ABB RobotStudio station: Proyecto.rsstn

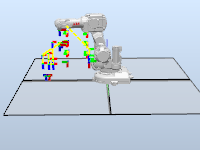
Station Proyecto (saved by RobotStudio 22.1.9826.0)
Controller IRB140_6_81
  mechanical unit ROB_1: IRB140_6_81_C_03_2, 6 joints, base frame (0, 0, 0) mm
Layout (positions relative to the parent item):
  - IRB140_6_81_C_03_2 [mechanism, from Robots\IRB140_6_81_C_G_03.rslib] at (0, 0, 0) mm; joint values [0.0983, 0.2535, -0.224, 0, 1.5413, 0.0983] (rad or m)
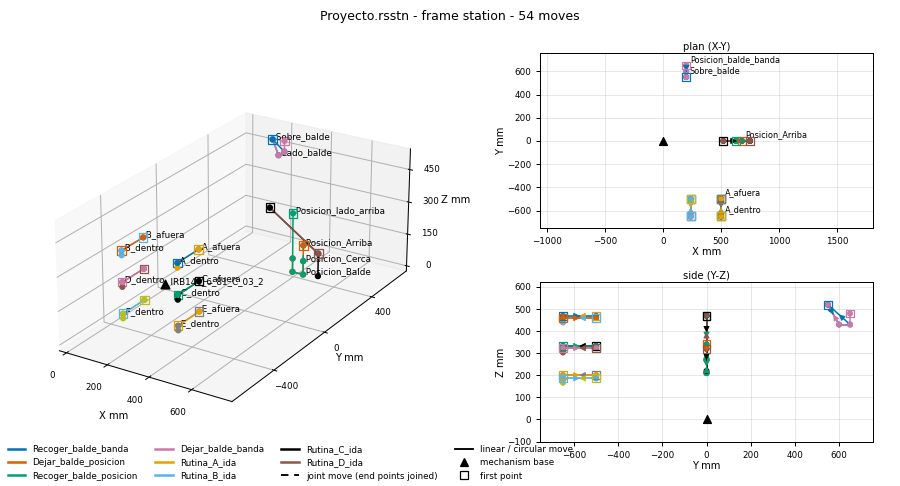
[picture p0: tool path of Proyecto.rsstn in frame station, 54 of 57 moves have a stored position in this frame; points joined in program order, loops and branches not executed]
Targets, tools, work objects and paths stored in the station, written as RAPID:
! task T_ROB1
MODULE Module1
  CONST jointtarget Home:=[[0,0,0,0,0,0],[9E+09,9E+09,9E+09,9E+09,9E+09,9E+09]];
  CONST robtarget Sobre_balde:=[[-100,0,-100],[0.707106781,0,0.707106781,0],[0,0,0,0],[9E+09,9E+09,9E+09,9E+09,9E+09,9E+09]];
  CONST robtarget Lado_balde:=[[-10,0,-50],[0.707106781,0,0.707106781,0],[0,0,-1,0],[9E+09,9E+09,9E+09,9E+09,9E+09,9E+09]];
  CONST robtarget Posicion_balde_banda:=[[-10,0,0],[0.707106781,0,0.707106781,0],[0,0,-1,0],[9E+09,9E+09,9E+09,9E+09,9E+09,9E+09]];
  CONST robtarget Dejando_balde:=[[-60,0,0],[0.707106781,0,0.707106781,0],[0,0,-1,0],[9E+09,9E+09,9E+09,9E+09,9E+09,9E+09]];
  CONST robtarget Posicion_Arriba:=[[-270,0,0],[0.707106781,0,0.707106781,0],[-1,1,-2,0],[9E+09,9E+09,9E+09,9E+09,9E+09,9E+09]];
  CONST robtarget Posicion_Cerca:=[[-200,0,0],[0.707106781,0,0.707106781,0],[-1,1,-2,0],[9E+09,9E+09,9E+09,9E+09,9E+09,9E+09]];
  CONST robtarget Posicion_Balde:=[[-140,0,0],[0.707106781,0,0.707106781,0],[-1,1,-2,0],[9E+09,9E+09,9E+09,9E+09,9E+09,9E+09]];
  CONST robtarget Posicion_lado:=[[-140,0,-50],[0.707106781,0,0.707106781,0],[-1,1,-2,0],[9E+09,9E+09,9E+09,9E+09,9E+09,9E+09]];
  CONST robtarget Posicion_lado_cerca:=[[-200,0,-50],[0.707106781,0,0.707106781,0],[0,0,0,0],[9E+09,9E+09,9E+09,9E+09,9E+09,9E+09]];
  CONST robtarget Posicion_lado_arriba:=[[-400,0,-50],[0.707106781,0,0.707106781,0],[0,0,0,0],[9E+09,9E+09,9E+09,9E+09,9E+09,9E+09]];
  CONST robtarget A_afuera:=[[-379,0,0],[1,0,0,0],[-1,0,-1,1],[9E+09,9E+09,9E+09,9E+09,9E+09,9E+09]];
  CONST robtarget A_dentro:=[[-379,0,150],[1,0,0,0],[-1,0,-1,1],[9E+09,9E+09,9E+09,9E+09,9E+09,9E+09]];
  CONST robtarget A_pieza:=[[-359,0,150],[1,0,0,0],[-1,0,-1,1],[9E+09,9E+09,9E+09,9E+09,9E+09,9E+09]];
  CONST robtarget B_afuera:=[[-369,-261,0],[1,0,0,0],[-1,0,-1,1],[9E+09,9E+09,9E+09,9E+09,9E+09,9E+09]];
  CONST robtarget B_dentro:=[[-369,-261,150],[1,0,0,0],[-1,0,-1,1],[9E+09,9E+09,9E+09,9E+09,9E+09,9E+09]];
  CONST robtarget B_pieza:=[[-349,-261,150],[1,0,0,0],[-1,0,-1,1],[9E+09,9E+09,9E+09,9E+09,9E+09,9E+09]];
  CONST robtarget C_afuera:=[[-243,0,0],[1,0,0,0],[-1,0,-1,1],[9E+09,9E+09,9E+09,9E+09,9E+09,9E+09]];
  CONST robtarget C_dentro:=[[-243,0,150],[1,0,0,0],[-1,0,-1,1],[9E+09,9E+09,9E+09,9E+09,9E+09,9E+09]];
  CONST robtarget C_pieza:=[[-223,0,150],[1,0,0,0],[-1,0,-1,1],[9E+09,9E+09,9E+09,9E+09,9E+09,9E+09]];
  CONST robtarget D_afuera:=[[-233,-261,0],[1,0,0,0],[-1,0,-1,1],[9E+09,9E+09,9E+09,9E+09,9E+09,9E+09]];
  CONST robtarget D_dentro:=[[-233,-261,150],[1,0,0,0],[-1,0,-1,1],[9E+09,9E+09,9E+09,9E+09,9E+09,9E+09]];
  CONST robtarget D_pieza:=[[-213,-261,150],[1,0,0,0],[-1,0,-1,1],[9E+09,9E+09,9E+09,9E+09,9E+09,9E+09]];
  CONST robtarget E_afuera:=[[-111,0,0],[1,0,0,0],[-1,0,-1,1],[9E+09,9E+09,9E+09,9E+09,9E+09,9E+09]];
  CONST robtarget E_dentro:=[[-111,0,150],[1,0,0,0],[-1,0,-1,1],[9E+09,9E+09,9E+09,9E+09,9E+09,9E+09]];
  CONST robtarget E_pieza:=[[-91,0,150],[1,0,0,0],[-1,0,-1,1],[9E+09,9E+09,9E+09,9E+09,9E+09,9E+09]];
  CONST robtarget F_afuera:=[[-96,-261,0],[1,0,0,0],[-1,0,0,1],[9E+09,9E+09,9E+09,9E+09,9E+09,9E+09]];
  CONST robtarget F_dentro:=[[-96,-261,150],[1,0,0,0],[-1,0,-1,1],[9E+09,9E+09,9E+09,9E+09,9E+09,9E+09]];
  CONST robtarget F_pieza:=[[-76,-261,150],[1,0,0,0],[-1,0,-1,1],[9E+09,9E+09,9E+09,9E+09,9E+09,9E+09]];
  CONST jointtarget Ac_repisa:=[[-27,44,-6,72,-69,-48],[9E+09,9E+09,9E+09,9E+09,9E+09,9E+09]];
  CONST robtarget Dejar_pieza:=[[-30,0,-150],[1,0,0,0],[0,0,0,0],[9E+09,9E+09,9E+09,9E+09,9E+09,9E+09]];
  CONST robtarget Sobre_pieza:=[[-30,0,-250],[1,0,0,0],[0,0,0,0],[9E+09,9E+09,9E+09,9E+09,9E+09,9E+09]];
  CONST robtarget Acercamiento_pieza:=[[200,0,-400],[1,0,0,0],[0,0,0,0],[9E+09,9E+09,9E+09,9E+09,9E+09,9E+09]];
  PROC Recoger_balde_banda()
    MoveAbsJ Home,v300,z100,Gancho\WObj:=Balde_banda;
    MoveJ Sobre_balde,v300,z100,Gancho\WObj:=Balde_banda;
    MoveL Lado_balde,v100,z100,Gancho\WObj:=Balde_banda;
    MoveL Posicion_balde_banda,v100,z100,Gancho\WObj:=Balde_banda;
    MoveL Sobre_balde,v100,z100,Gancho\WObj:=Balde_banda;
  ENDPROC
  PROC Dejar_balde_posicion()
    MoveL Posicion_Arriba,v100,z100,Gancho\WObj:=Balde_posicion;
    MoveL Posicion_Cerca,v100,z100,Gancho\WObj:=Balde_posicion;
    MoveL Posicion_Balde,v100,z100,Gancho\WObj:=Balde_posicion;
    MoveL Posicion_lado,v100,z100,Gancho\WObj:=Balde_posicion;
    MoveL Posicion_lado_cerca,v100,z100,Gancho\WObj:=Balde_posicion;
  ENDPROC
  PROC Recoger_balde_posicion()
    MoveL Posicion_lado_arriba,v300,z100,Gancho\WObj:=Balde_posicion;
    MoveL Posicion_lado_cerca,v300,z100,Gancho\WObj:=Balde_posicion;
    MoveL Posicion_lado,v100,z100,Gancho\WObj:=Balde_posicion;
    MoveL Posicion_Balde,v100,z100,Gancho\WObj:=Balde_posicion;
    MoveL Posicion_Cerca,v100,z100,Gancho\WObj:=Balde_posicion;
    MoveJ Posicion_Arriba,v100,z100,Gancho\WObj:=Balde_posicion;
  ENDPROC
  PROC Dejar_balde_banda()
    MoveL Dejando_balde,v100,z100,Gancho\WObj:=Balde_banda;
    MoveL Posicion_balde_banda,v100,z100,Gancho\WObj:=Balde_banda;
    MoveL Lado_balde,v100,z100,Gancho\WObj:=Balde_banda;
    MoveL Sobre_balde,v100,z100,Gancho\WObj:=Balde_banda;
  ENDPROC
  PROC Rutina_A_ida()
    MoveL A_afuera,v300,z100,Ventosa\WObj:=Repisa;
    MoveL A_dentro,v300,z100,Ventosa\WObj:=Repisa;
    MoveL A_pieza,v300,z100,Ventosa\WObj:=Repisa;
  ENDPROC
  PROC Rutina_B_ida()
    MoveL B_afuera,v300,z100,Ventosa\WObj:=Repisa;
    MoveL B_dentro,v300,z100,Ventosa\WObj:=Repisa;
    MoveL B_pieza,v300,z100,Ventosa\WObj:=Repisa;
  ENDPROC
  PROC Rutina_C_ida()
    MoveL C_afuera,v300,z100,Ventosa\WObj:=Repisa;
    MoveL C_dentro,v300,z100,Ventosa\WObj:=Repisa;
    MoveL C_pieza,v300,z100,Ventosa\WObj:=Repisa;
  ENDPROC
  PROC Rutina_D_ida()
    MoveL D_afuera,v300,z100,Ventosa\WObj:=Repisa;
    MoveL D_dentro,v300,z100,Ventosa\WObj:=Repisa;
    MoveL D_pieza,v300,z100,Ventosa\WObj:=Repisa;
  ENDPROC
  PROC Rutina_E_ida()
    MoveL E_afuera,v300,z100,Ventosa\WObj:=Repisa;
    MoveL E_dentro,v300,z100,Ventosa\WObj:=Repisa;
    MoveL E_pieza,v300,z100,Ventosa\WObj:=Repisa;
  ENDPROC
  PROC Rutina_F_ida()
    MoveL F_afuera,v300,z100,Ventosa\WObj:=Repisa;
    MoveL F_dentro,v300,z100,Ventosa\WObj:=Repisa;
    MoveL F_pieza,v300,z100,Ventosa\WObj:=Repisa;
  ENDPROC
  PROC Rutina_A_regreso()
    MoveL A_dentro,v300,z100,Ventosa\WObj:=Repisa;
    MoveL A_afuera,v300,z100,Ventosa\WObj:=Repisa;
  ENDPROC
  PROC Rutina_B_regreso()
    MoveL B_dentro,v300,z100,Ventosa\WObj:=Repisa;
    MoveL B_afuera,v300,z100,Ventosa\WObj:=Repisa;
  ENDPROC
  PROC Rutina_C_regreso()
    MoveL C_dentro,v300,z100,Ventosa\WObj:=Repisa;
    MoveL C_afuera,v300,z100,Ventosa\WObj:=Repisa;
  ENDPROC
  PROC Rutina_D_regreso()
    MoveL D_dentro,v300,z100,Ventosa\WObj:=Repisa;
    MoveL D_afuera,v300,z100,Ventosa\WObj:=Repisa;
  ENDPROC
  PROC Rutina_E_regreso()
    MoveL E_dentro,v300,z100,Ventosa\WObj:=Repisa;
    MoveL E_afuera,v300,z100,Ventosa\WObj:=Repisa;
  ENDPROC
  PROC Rutina_F_regreso()
    MoveL F_dentro,v300,z100,Ventosa\WObj:=Repisa;
    MoveL F_afuera,v300,z100,Ventosa\WObj:=Repisa;
  ENDPROC
  PROC Pieza_Dejar_ida()
    MoveJ Acercamiento_pieza,v300,z100,Ventosa\WObj:=Balde_pieza;
    MoveL Sobre_pieza,v300,z100,Ventosa\WObj:=Balde_pieza;
    MoveL Dejar_pieza,v300,z100,Ventosa\WObj:=Balde_pieza;
  ENDPROC
  PROC Pieza_Dejar_Regreso()
    MoveL Sobre_pieza,v300,z100,Ventosa\WObj:=Balde_pieza;
    MoveL Acercamiento_pieza,v300,z100,Ventosa\WObj:=Balde_pieza;
  ENDPROC
  PROC Ir_estanteria()
    MoveAbsJ Ac_repisa,v300,z100,Ventosa\WObj:=Balde_pieza;
  ENDPROC
  PROC Ir_home()
    MoveAbsJ Home,v300,z100,Ventosa\WObj:=Balde_pieza;
  ENDPROC
ENDMODULE

! task T_ROB1
MODULE CalibData
  TASK PERS tooldata Gancho:=[TRUE,[[0,60.02,164.11],[1,0,0,0]],[1,[0,0,1],[1,0,0,0],0,0,0]];
  TASK PERS tooldata Ventosa:=[TRUE,[[17.5,-53,154.3],[1,0,0,0]],[1,[0,0,1],[1,0,0,0],0,0,0]];
  TASK PERS wobjdata Balde_banda:=[FALSE,TRUE,"",[[200,650,420],[0.5,-0.5,0.5,0.5]],[[0,0,0],[1,0,0,0]]];
  TASK PERS wobjdata Balde_posicion:=[FALSE,TRUE,"",[[680,0,70],[0.707106781,0,0.707106781,0]],[[0,0,0],[1,0,0,0]]];
  TASK PERS wobjdata Repisa:=[FALSE,TRUE,"",[[500,-500,90],[0.5,0.5,0.5,-0.5]],[[0,0,0],[1,0,0,0]]];
  TASK PERS wobjdata Balde_pieza:=[FALSE,TRUE,"",[[720,0,70],[0,0,1,0]],[[0,0,0],[1,0,0,0]]];
ENDMODULE

